RoboDK station: cable_bending.rdk

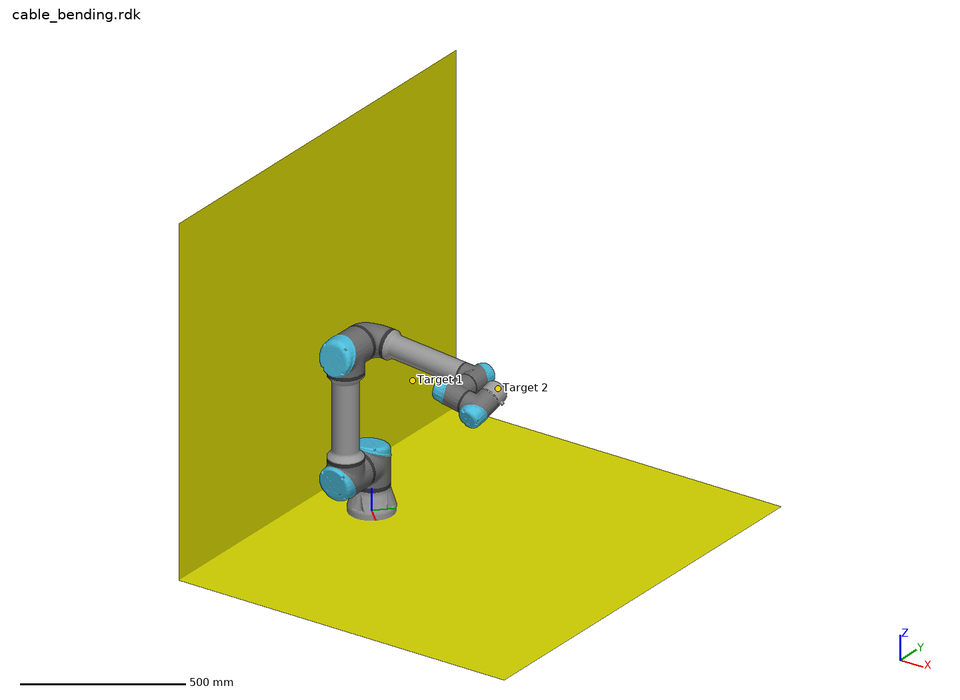
[picture v0: the station drawn from its stored meshes, robots at their saved joint values, targets as dots, program paths as lines]
Station cable_bending. Poses are relative to the parent item; angles as X-Y-Z fixed-axis rotations.
Station parameters (name, value as stored): CollisionFreePlanner, UR5e, CollisionFreePlanner-Rob UR5e
  - frame UR5e Base at (0, 0, 0) mm, rotated rx 0 ry 0 rz -45 deg
    - robot UR5e: 6 axes, payload 5 kg, reach 850 mm, repeatability 0.03 mm, weight 18.4 kg
        modified DH rows (alpha deg, a mm, theta deg, d mm): 0, 0, 0, 162.5; 90, 0, 180, 0; 0, 425, 0, 0; 0, 392.25, 0, 133.3; -90, 0, 0, 99.7; 90, 0, 180, 99.6
        joint limits [-360, -360, -360, -360, -360, -360] to [360, 360, 360, 360, 360, 360]; home [0, -90, -90, 0, 90, 0]; saved at [44.99, -90, -95.33, -96.68, -161.13, 19.18]
    - target Target 1 (joint target) at (386.71, 57.43, 615.38) mm, rotated rx -82.99 ry 71.71 rz -126.68 deg; joints [44.99, -89.99, -95.33, 58.01, 2.76, 19.18] of UR5e
    - target Target 2 (joint target) at (377.53, 322.18, 561.83) mm, rotated rx 57.71 ry 53.69 rz -166.06 deg; joints [44.99, -90, -95.33, -96.68, -161.13, 19.18] of UR5e
  - object Right wall at (0, 0, 0) mm, size 1200 x 1200 x 0.6 mm, geometry from plane_1m.sld
  - object Floor at (0, 0, 0) mm, size 1200 x 1460 x 0.6 mm
  - object Left wall at (0, 0, 0) mm, size 1200 x 1200 x 0.6 mm, geometry from plane_1m.sld
  - object Back wall at (0, 0, 0) mm, rotated rx 0 ry -90 rz 0 deg, size 1200 x 1460 x 0.6 mm
  - object Front wall at (0, 0, 0) mm, rotated rx 0 ry -90 rz 0 deg, size 1200 x 1460 x 0.6 mm
  - Python program roboDK_test (listed below)

--- Python program roboDK_test ---
from robolink import *
from robodk import *
from datetime import datetime

timestamp = datetime.now()
filename = "cycle_count_" + timestamp.strftime("%d_%m_%Y_%H_%M_%S")+".txt"
path = "/home/melyso/Documents/python_scripts/cycle_counts/" + filename
fo = open(path, "w")
fo.write("0")
fo.close()

RDK = Robolink()
robot = RDK.Item('UR5e', ITEM_TYPE_ROBOT)
target_1 = RDK.Item('Target 1')
target_2 = RDK.Item('Target 2')


robot.MoveJ(target_1)

while True:
	robot.MoveJ(target_2)
	robot.MoveJ(target_1)
	fo = open(path, "r")
	cycle_count = int(fo.read())
	fo.close()
	cycle_count += 1
	fo = open(path, "w")
	fo.write(str(cycle_count))
	fo.close()
	print("Cycles performed: ", cycle_count)
